PROGRAM MAIN
VAR
END_VAR

END_PROGRAM

(* stored: Version 1.1.0.1
   POU MAIN: Id {dc49c998-00cd-4be4-93d5-341d399a0e32} *)
